FUNCTION_BLOCK FB_FSS2_WriteFileForGMES
VAR_INPUT
	bExecute			: BOOL;			(* scan for valid Outer in arrOuterStatus *)
	strLocalCHMPath					: STRING(255);
	strGMESFile						: T_CHM_Filename;
	nOutersPerCase						: UINT;
END_VAR
VAR_IN_OUT
	stAgregationData	 			: ST_CHM_Data;		(* case data to be written to XML *)
END_VAR
VAR_OUTPUT
	bDone				: BOOL;			(* TRUE = write OAC file complete *)
	bBusy				: BOOL;			(* TRUE = write OAC file in progress *)
	bError				: BOOL;			(* TRUE = write OAC file error *)
	nErrorID			: UDINT;		(* error ID *)
	nImigeProcessingSize				:UDINT;
END_VAR
VAR
	fbExecute			: R_TRIG;
	eState				: E_XML_CtrlState;
	eErrorState			: E_XML_CtrlState;

	fbBuildGMESData		: FB_FSS2_BuildXMLDataForGMES;
	fbWriteFile			: FB_FILE_WriteByByte;
END_VAR

(* monitor bExecute for rising edge *)
fbExecute(CLK := bExecute);

CASE eState OF

	(* idle *)
	E_XML_IDLE:

		(* rising edge on bExecute *)
		IF fbExecute.Q = TRUE THEN

			(* update outputs *)
			bDone := FALSE;
			bBusy := TRUE;
			bError := FALSE;
			nErrorID := 0;

			eErrorState := eState;

			(* generate XML file name and clear data for last XML file *)

			strGMESFile := F_CONCAT3('GMES_','XXXXXXXXX', '.xml');

			eState := E_XML_GENERATEIMAGE;

		(* disabled *)
		ELSIF bExecute = FALSE THEN

			(* update outputs *)
			bDone := FALSE;
			bBusy := FALSE;
			bError := FALSE;
			nErrorID := 0;
		END_IF


	(* build  image in XML format *)
	E_XML_GENERATEIMAGE:

		(* build XML data *)
		fbBuildGMESData(
			bExecute		:= TRUE,
			nCartonsPerMasterCase	:=nOutersPerCase,
			stAgregationData := stAgregationData
		);

		(* build XML data complete *)
		IF fbBuildGMESData.bDone = TRUE THEN

			eState := E_XML_WRITEXML;
			nImigeProcessingSize	:= fbBuildGMESData.nImageByte;

			(* close off fbBuildXMLData *)
			fbBuildGMESData(bExecute := FALSE, stAgregationData := stAgregationData);
		END_IF


	(* write XML image *)
	E_XML_WRITEXML:

		(* write XML template to file *)
		fbWriteFile(
			bExecute	:= TRUE,
			pSourceAddr	:= ADR(fbBuildGMESData.arrXMLImage),
			nSourceSize	:= fbBuildGMESData.nImageByte,
			strPathFile	:= CONCAT(strLocalCHMPath, strGMESFile),
			tTimeout	:= T#1s
		);

		(* file write complete *)
		IF fbWriteFile.bDone = TRUE THEN

			(* file write completed OK *)
			IF fbWriteFile.bError = FALSE THEN

				;

			(* file write error *)
			ELSE

				bError := TRUE;
				nErrorID := fbWriteFile.nErrorID;
				eErrorState := eState;
			END_IF

			eState := E_XML_DONE;

			(* close of fbWriteFile *)
			fbWriteFile(bExecute := FALSE);
		END_IF


	(* XML file complete *)
	E_XML_DONE:

		(* update outputs *)
		bDone := TRUE;
		bBusy := FALSE;

		eState := E_XML_IDLE;


(* unknown state *)
ELSE

	eState := E_XML_IDLE;
END_CASE

END_FUNCTION_BLOCK

(* stored: Version 1.1.0.1, ProductVersion 3.1.4024.15
   POU FB_FSS2_WriteFileForGMES: Id {c28f18a3-0a5c-4f5a-8636-98a7019d83ac}, SpecialFunc None *)
